% RSLogix 500 project Grain Separator - Onsite 24-11-05.RSS, saved by version 6.30.00.12 %
PROJECT "CORSON1"    % processor: SLC 500, 1747-L532 %

PROGRAM FILES
  LAD 2   10 rungs
  LAD 4   19 rungs
  LAD 5   124 rungs
  LAD 6   61 rungs
  LAD 7   60 rungs
  LAD 8   20 rungs
  LAD 9   20 rungs
  LAD 10   62 rungs
  LAD 11   79 rungs

DATA FILES
  O0 OUTPUT  11 elements
  I1 INPUT  11 elements
  S2 STATUS  83 elements
  B3 BINARY  1 elements
  T4 TIMER  1 elements
  C5 COUNTER  1 elements
  R6 CONTROL  1 elements
  N7 INTEGER  1 elements
  F8 FLOAT  1 elements
  B9   1 elements
  B10   2 elements
  T11   10 elements
  N12   1 elements
  B13   14 elements
  T14   60 elements
  N15   10 elements
  B16   5 elements
  T17   60 elements
  N18   1 elements
  B19   5 elements
  T20   60 elements
  N21   1 elements
  B22   5 elements
  T23   17 elements
  N24   1 elements
  B25   5 elements
  T26   16 elements
  N27   1 elements
  B28   1 elements
  T29   13 elements
  N30   1 elements
  B31   1 elements

LADDER 2
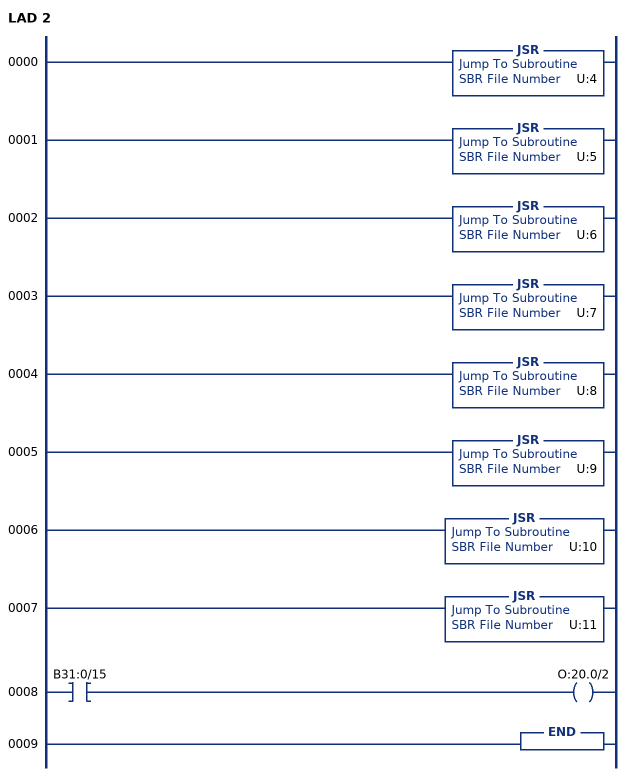
% Rung: 0 %
SOR JSR U:4 EOR
% Rung: 1 %
SOR JSR U:5 EOR
% Rung: 2 %
SOR JSR U:6 EOR
% Rung: 3 %
SOR JSR U:7 EOR
% Rung: 4 %
SOR JSR U:8 EOR
% Rung: 5 %
SOR JSR U:9 EOR
% Rung: 6 %
SOR JSR U:10 EOR
% Rung: 7 %
SOR JSR U:11 EOR
% Rung: 8 %
SOR XIC B31:0/15 OTE O:20.0/2 EOR
% Rung: 9 %
SOR END EOR

LADDER 4
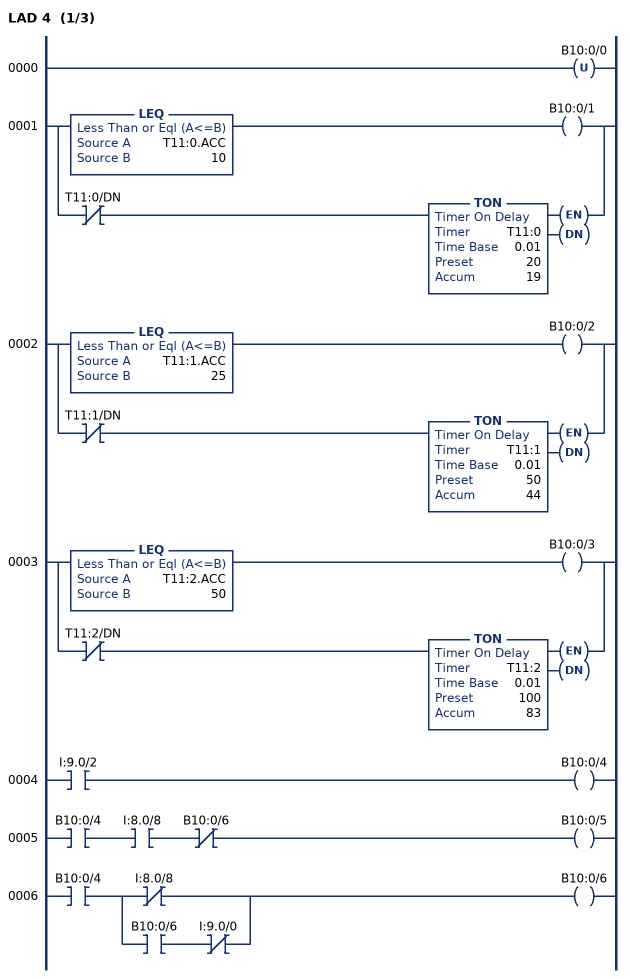
% Rung: 0 %
SOR OTU B10:0/0 EOR
% Rung: 1 %
SOR BST LEQ T11:0.ACC 10 OTE B10:0/1 NXB XIO T11:0/DN TON T11:0 0.01 20 19 BND EOR
% Rung: 2 %
SOR BST LEQ T11:1.ACC 25 OTE B10:0/2 NXB XIO T11:1/DN TON T11:1 0.01 50 44 BND EOR
% Rung: 3 %
SOR BST LEQ T11:2.ACC 50 OTE B10:0/3 NXB XIO T11:2/DN TON T11:2 0.01 100 83 BND EOR
% Rung: 4 %
SOR XIC I:9.0/2 OTE B10:0/4 EOR
% Rung: 5 %
SOR XIC B10:0/4 XIC I:8.0/8 XIO B10:0/6 OTE B10:0/5 EOR
% Rung: 6 %
SOR XIC B10:0/4 BST XIO I:8.0/8 NXB XIC B10:0/6 XIO I:9.0/0 BND OTE B10:0/6 EOR

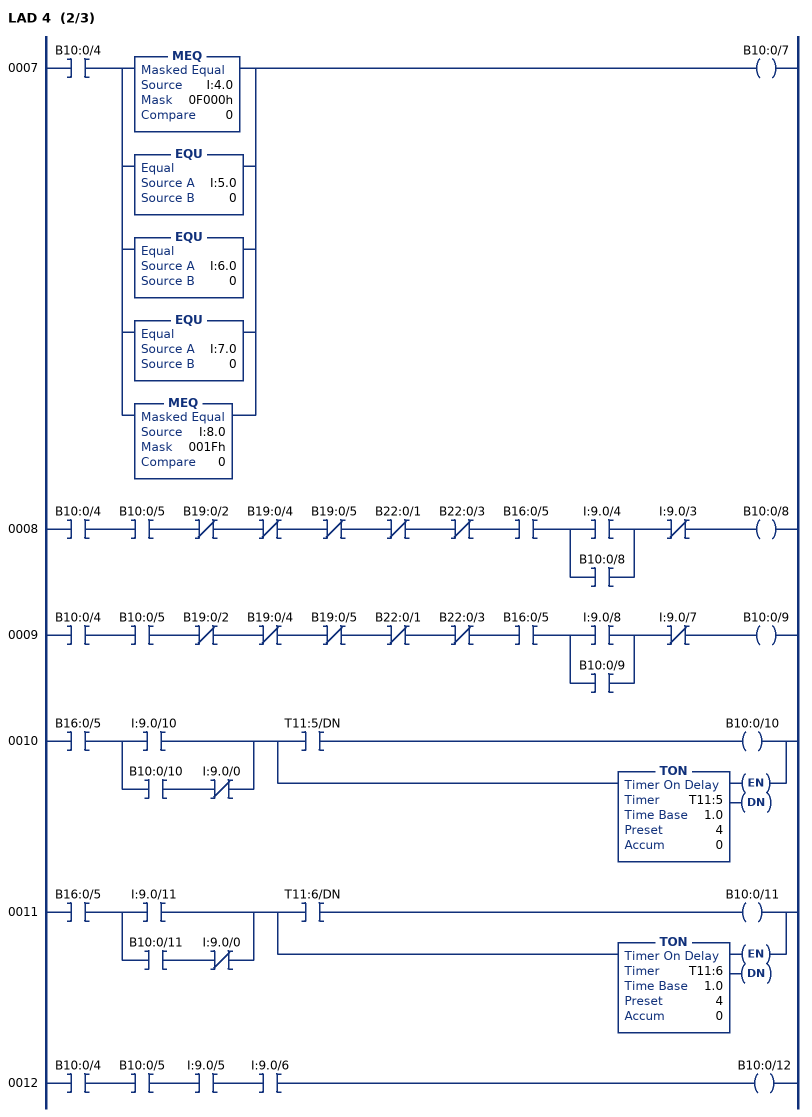
% Rung: 7 %
SOR XIC B10:0/4 BST MEQ I:4.0 0F000h 0 NXB EQU I:5.0 0 NXB EQU I:6.0 0 NXB EQU I:7.0 0 NXB MEQ I:8.0 001Fh 0 BND OTE B10:0/7 EOR
% Rung: 8 %
SOR XIC B10:0/4 XIC B10:0/5 XIO B19:0/2 XIO B19:0/4 XIO B19:0/5 XIO B22:0/1 XIO B22:0/3 XIC B16:0/5 BST XIC I:9.0/4 NXB XIC B10:0/8 BND XIO I:9.0/3 OTE B10:0/8 EOR
% Rung: 9 %
SOR XIC B10:0/4 XIC B10:0/5 XIO B19:0/2 XIO B19:0/4 XIO B19:0/5 XIO B22:0/1 XIO B22:0/3 XIC B16:0/5 BST XIC I:9.0/8 NXB XIC B10:0/9 BND XIO I:9.0/7 OTE B10:0/9 EOR
% Rung: 10 %
SOR XIC B16:0/5 BST XIC I:9.0/10 NXB XIC B10:0/10 XIO I:9.0/0 BND BST XIC T11:5/DN OTE B10:0/10 NXB TON T11:5 1.0 4 0 BND EOR
% Rung: 11 %
SOR XIC B16:0/5 BST XIC I:9.0/11 NXB XIC B10:0/11 XIO I:9.0/0 BND BST XIC T11:6/DN OTE B10:0/11 NXB TON T11:6 1.0 4 0 BND EOR
% Rung: 12 %
SOR XIC B10:0/4 XIC B10:0/5 XIC I:9.0/5 XIC I:9.0/6 OTE B10:0/12 EOR

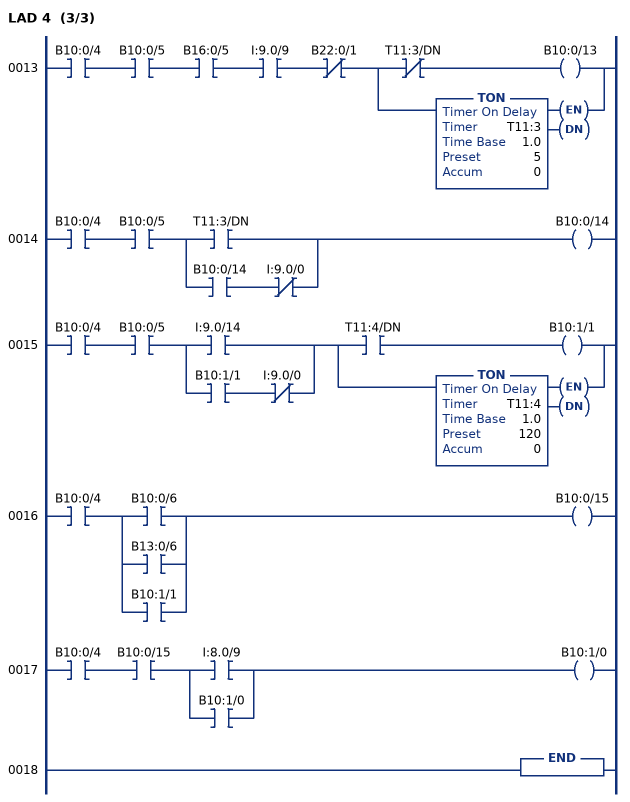
% Rung: 13 %
SOR XIC B10:0/4 XIC B10:0/5 XIC B16:0/5 XIC I:9.0/9 XIO B22:0/1 BST XIO T11:3/DN OTE B10:0/13 NXB TON T11:3 1.0 5 0 BND EOR
% Rung: 14 %
SOR XIC B10:0/4 XIC B10:0/5 BST XIC T11:3/DN NXB XIC B10:0/14 XIO I:9.0/0 BND OTE B10:0/14 EOR
% Rung: 15 %
SOR XIC B10:0/4 XIC B10:0/5 BST XIC I:9.0/14 NXB XIC B10:1/1 XIO I:9.0/0 BND BST XIC T11:4/DN OTE B10:1/1 NXB TON T11:4 1.0 120 0 BND EOR
% Rung: 16 %
SOR XIC B10:0/4 BST XIC B10:0/6 NXB XIC B13:0/6 NXB XIC B10:1/1 BND OTE B10:0/15 EOR
% Rung: 17 %
SOR XIC B10:0/4 XIC B10:0/15 BST XIC I:8.0/9 NXB XIC B10:1/0 BND OTE B10:1/0 EOR
% Rung: 18 %
SOR END EOR

LADDER 5
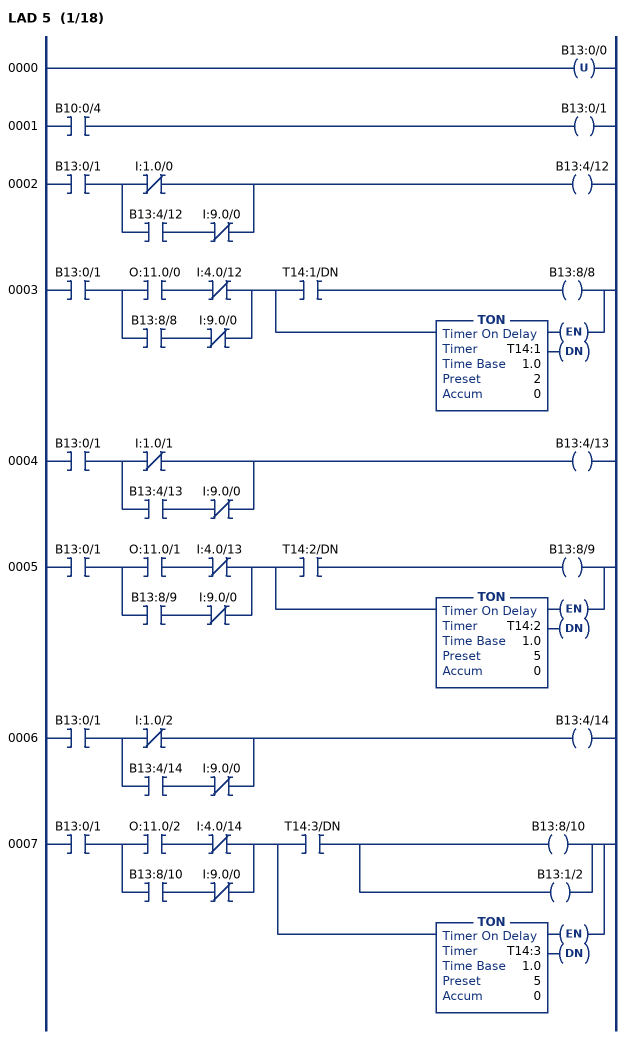
% Rung: 0 %
SOR OTU B13:0/0 EOR
% Rung: 1 %
SOR XIC B10:0/4 OTE B13:0/1 EOR
% Rung: 2 %
SOR XIC B13:0/1 BST XIO I:1.0/0 NXB XIC B13:4/12 XIO I:9.0/0 BND OTE B13:4/12 EOR
% Rung: 3 %
SOR XIC B13:0/1 BST XIC O:11.0/0 XIO I:4.0/12 NXB XIC B13:8/8 XIO I:9.0/0 BND BST XIC T14:1/DN OTE B13:8/8 NXB TON T14:1 1.0 2 0 BND EOR
% Rung: 4 %
SOR XIC B13:0/1 BST XIO I:1.0/1 NXB XIC B13:4/13 XIO I:9.0/0 BND OTE B13:4/13 EOR
% Rung: 5 %
SOR XIC B13:0/1 BST XIC O:11.0/1 XIO I:4.0/13 NXB XIC B13:8/9 XIO I:9.0/0 BND BST XIC T14:2/DN OTE B13:8/9 NXB TON T14:2 1.0 5 0 BND EOR
% Rung: 6 %
SOR XIC B13:0/1 BST XIO I:1.0/2 NXB XIC B13:4/14 XIO I:9.0/0 BND OTE B13:4/14 EOR
% Rung: 7 %
SOR XIC B13:0/1 BST XIC O:11.0/2 XIO I:4.0/14 NXB XIC B13:8/10 XIO I:9.0/0 BND BST XIC T14:3/DN BST OTE B13:8/10 NXB OTE B13:1/2 BND NXB TON T14:3 1.0 5 0 BND EOR

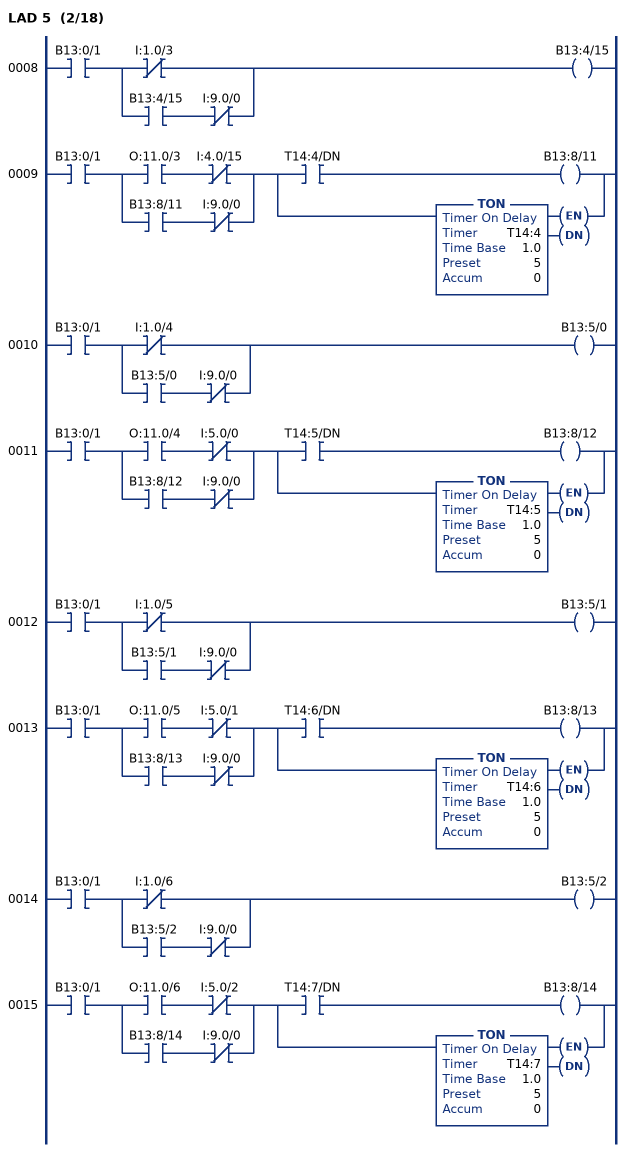
% Rung: 8 %
SOR XIC B13:0/1 BST XIO I:1.0/3 NXB XIC B13:4/15 XIO I:9.0/0 BND OTE B13:4/15 EOR
% Rung: 9 %
SOR XIC B13:0/1 BST XIC O:11.0/3 XIO I:4.0/15 NXB XIC B13:8/11 XIO I:9.0/0 BND BST XIC T14:4/DN OTE B13:8/11 NXB TON T14:4 1.0 5 0 BND EOR
% Rung: 10 %
SOR XIC B13:0/1 BST XIO I:1.0/4 NXB XIC B13:5/0 XIO I:9.0/0 BND OTE B13:5/0 EOR
% Rung: 11 %
SOR XIC B13:0/1 BST XIC O:11.0/4 XIO I:5.0/0 NXB XIC B13:8/12 XIO I:9.0/0 BND BST XIC T14:5/DN OTE B13:8/12 NXB TON T14:5 1.0 5 0 BND EOR
% Rung: 12 %
SOR XIC B13:0/1 BST XIO I:1.0/5 NXB XIC B13:5/1 XIO I:9.0/0 BND OTE B13:5/1 EOR
% Rung: 13 %
SOR XIC B13:0/1 BST XIC O:11.0/5 XIO I:5.0/1 NXB XIC B13:8/13 XIO I:9.0/0 BND BST XIC T14:6/DN OTE B13:8/13 NXB TON T14:6 1.0 5 0 BND EOR
% Rung: 14 %
SOR XIC B13:0/1 BST XIO I:1.0/6 NXB XIC B13:5/2 XIO I:9.0/0 BND OTE B13:5/2 EOR
% Rung: 15 %
SOR XIC B13:0/1 BST XIC O:11.0/6 XIO I:5.0/2 NXB XIC B13:8/14 XIO I:9.0/0 BND BST XIC T14:7/DN OTE B13:8/14 NXB TON T14:7 1.0 5 0 BND EOR

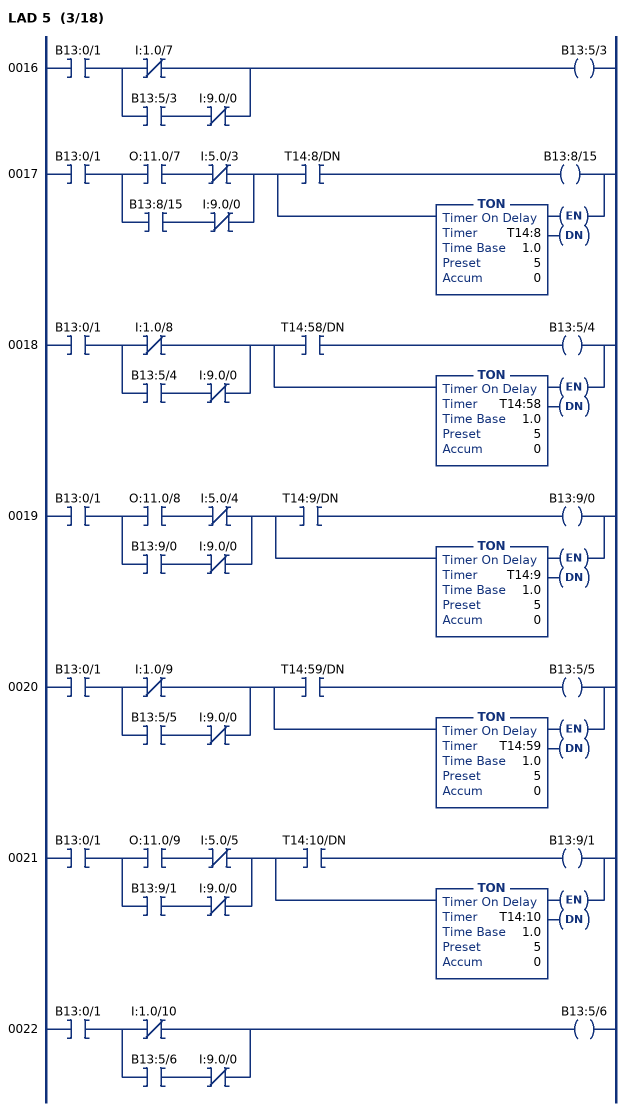
% Rung: 16 %
SOR XIC B13:0/1 BST XIO I:1.0/7 NXB XIC B13:5/3 XIO I:9.0/0 BND OTE B13:5/3 EOR
% Rung: 17 %
SOR XIC B13:0/1 BST XIC O:11.0/7 XIO I:5.0/3 NXB XIC B13:8/15 XIO I:9.0/0 BND BST XIC T14:8/DN OTE B13:8/15 NXB TON T14:8 1.0 5 0 BND EOR
% Rung: 18 %
SOR XIC B13:0/1 BST XIO I:1.0/8 NXB XIC B13:5/4 XIO I:9.0/0 BND BST XIC T14:58/DN OTE B13:5/4 NXB TON T14:58 1.0 5 0 BND EOR
% Rung: 19 %
SOR XIC B13:0/1 BST XIC O:11.0/8 XIO I:5.0/4 NXB XIC B13:9/0 XIO I:9.0/0 BND BST XIC T14:9/DN OTE B13:9/0 NXB TON T14:9 1.0 5 0 BND EOR
% Rung: 20 %
SOR XIC B13:0/1 BST XIO I:1.0/9 NXB XIC B13:5/5 XIO I:9.0/0 BND BST XIC T14:59/DN OTE B13:5/5 NXB TON T14:59 1.0 5 0 BND EOR
% Rung: 21 %
SOR XIC B13:0/1 BST XIC O:11.0/9 XIO I:5.0/5 NXB XIC B13:9/1 XIO I:9.0/0 BND BST XIC T14:10/DN OTE B13:9/1 NXB TON T14:10 1.0 5 0 BND EOR
% Rung: 22 %
SOR XIC B13:0/1 BST XIO I:1.0/10 NXB XIC B13:5/6 XIO I:9.0/0 BND OTE B13:5/6 EOR

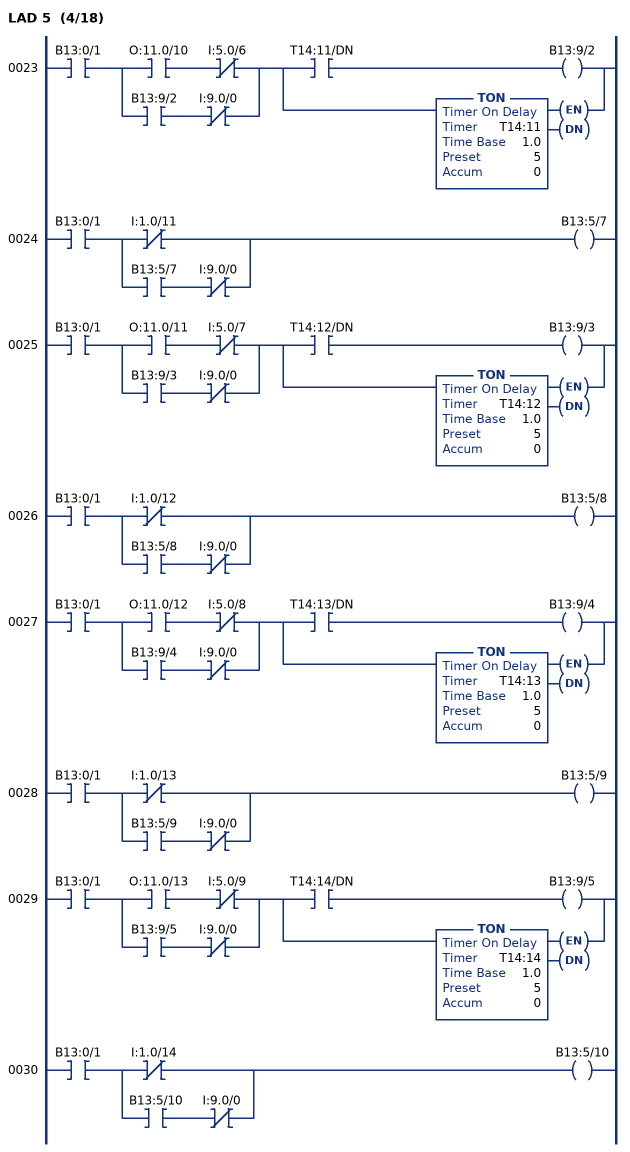
% Rung: 23 %
SOR XIC B13:0/1 BST XIC O:11.0/10 XIO I:5.0/6 NXB XIC B13:9/2 XIO I:9.0/0 BND BST XIC T14:11/DN OTE B13:9/2 NXB TON T14:11 1.0 5 0 BND EOR
% Rung: 24 %
SOR XIC B13:0/1 BST XIO I:1.0/11 NXB XIC B13:5/7 XIO I:9.0/0 BND OTE B13:5/7 EOR
% Rung: 25 %
SOR XIC B13:0/1 BST XIC O:11.0/11 XIO I:5.0/7 NXB XIC B13:9/3 XIO I:9.0/0 BND BST XIC T14:12/DN OTE B13:9/3 NXB TON T14:12 1.0 5 0 BND EOR
% Rung: 26 %
SOR XIC B13:0/1 BST XIO I:1.0/12 NXB XIC B13:5/8 XIO I:9.0/0 BND OTE B13:5/8 EOR
% Rung: 27 %
SOR XIC B13:0/1 BST XIC O:11.0/12 XIO I:5.0/8 NXB XIC B13:9/4 XIO I:9.0/0 BND BST XIC T14:13/DN OTE B13:9/4 NXB TON T14:13 1.0 5 0 BND EOR
% Rung: 28 %
SOR XIC B13:0/1 BST XIO I:1.0/13 NXB XIC B13:5/9 XIO I:9.0/0 BND OTE B13:5/9 EOR
% Rung: 29 %
SOR XIC B13:0/1 BST XIC O:11.0/13 XIO I:5.0/9 NXB XIC B13:9/5 XIO I:9.0/0 BND BST XIC T14:14/DN OTE B13:9/5 NXB TON T14:14 1.0 5 0 BND EOR
% Rung: 30 %
SOR XIC B13:0/1 BST XIO I:1.0/14 NXB XIC B13:5/10 XIO I:9.0/0 BND OTE B13:5/10 EOR

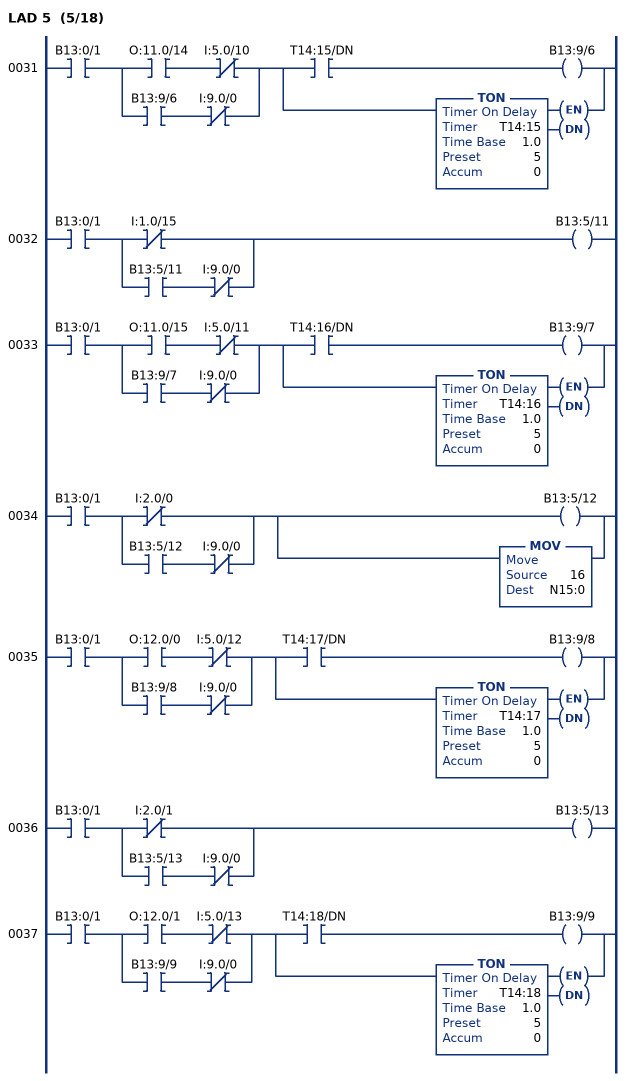
% Rung: 31 %
SOR XIC B13:0/1 BST XIC O:11.0/14 XIO I:5.0/10 NXB XIC B13:9/6 XIO I:9.0/0 BND BST XIC T14:15/DN OTE B13:9/6 NXB TON T14:15 1.0 5 0 BND EOR
% Rung: 32 %
SOR XIC B13:0/1 BST XIO I:1.0/15 NXB XIC B13:5/11 XIO I:9.0/0 BND OTE B13:5/11 EOR
% Rung: 33 %
SOR XIC B13:0/1 BST XIC O:11.0/15 XIO I:5.0/11 NXB XIC B13:9/7 XIO I:9.0/0 BND BST XIC T14:16/DN OTE B13:9/7 NXB TON T14:16 1.0 5 0 BND EOR
% Rung: 34 %
SOR XIC B13:0/1 BST XIO I:2.0/0 NXB XIC B13:5/12 XIO I:9.0/0 BND BST OTE B13:5/12 NXB MOV 16 N15:0 BND EOR
% Rung: 35 %
SOR XIC B13:0/1 BST XIC O:12.0/0 XIO I:5.0/12 NXB XIC B13:9/8 XIO I:9.0/0 BND BST XIC T14:17/DN OTE B13:9/8 NXB TON T14:17 1.0 5 0 BND EOR
% Rung: 36 %
SOR XIC B13:0/1 BST XIO I:2.0/1 NXB XIC B13:5/13 XIO I:9.0/0 BND OTE B13:5/13 EOR
% Rung: 37 %
SOR XIC B13:0/1 BST XIC O:12.0/1 XIO I:5.0/13 NXB XIC B13:9/9 XIO I:9.0/0 BND BST XIC T14:18/DN OTE B13:9/9 NXB TON T14:18 1.0 5 0 BND EOR

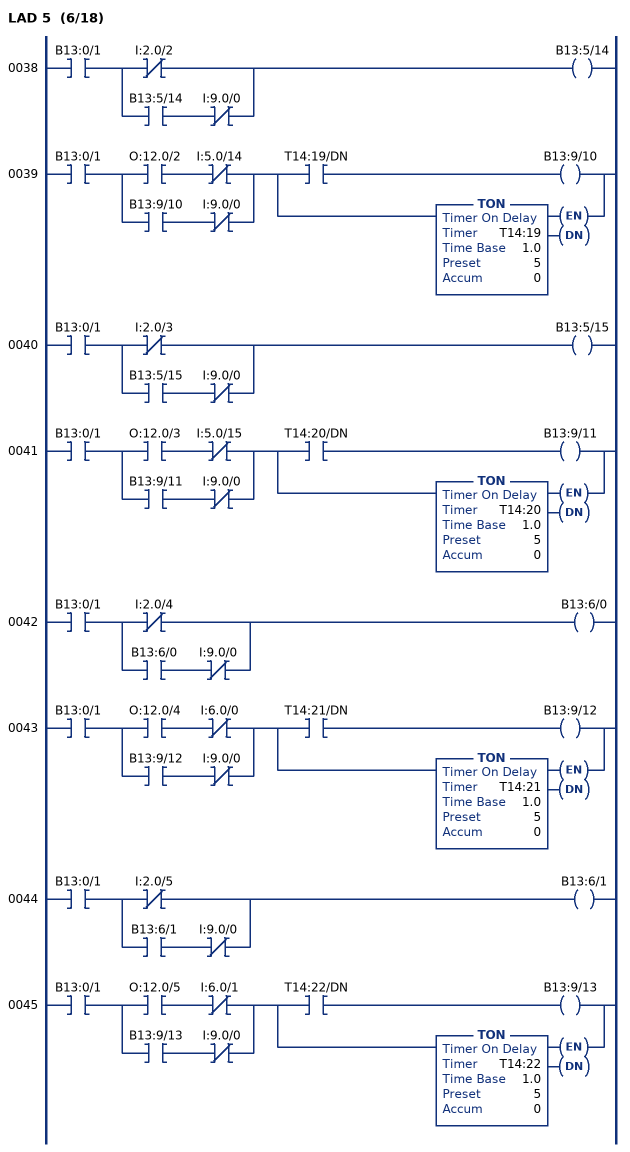
% Rung: 38 %
SOR XIC B13:0/1 BST XIO I:2.0/2 NXB XIC B13:5/14 XIO I:9.0/0 BND OTE B13:5/14 EOR
% Rung: 39 %
SOR XIC B13:0/1 BST XIC O:12.0/2 XIO I:5.0/14 NXB XIC B13:9/10 XIO I:9.0/0 BND BST XIC T14:19/DN OTE B13:9/10 NXB TON T14:19 1.0 5 0 BND EOR
% Rung: 40 %
SOR XIC B13:0/1 BST XIO I:2.0/3 NXB XIC B13:5/15 XIO I:9.0/0 BND OTE B13:5/15 EOR
% Rung: 41 %
SOR XIC B13:0/1 BST XIC O:12.0/3 XIO I:5.0/15 NXB XIC B13:9/11 XIO I:9.0/0 BND BST XIC T14:20/DN OTE B13:9/11 NXB TON T14:20 1.0 5 0 BND EOR
% Rung: 42 %
SOR XIC B13:0/1 BST XIO I:2.0/4 NXB XIC B13:6/0 XIO I:9.0/0 BND OTE B13:6/0 EOR
% Rung: 43 %
SOR XIC B13:0/1 BST XIC O:12.0/4 XIO I:6.0/0 NXB XIC B13:9/12 XIO I:9.0/0 BND BST XIC T14:21/DN OTE B13:9/12 NXB TON T14:21 1.0 5 0 BND EOR
% Rung: 44 %
SOR XIC B13:0/1 BST XIO I:2.0/5 NXB XIC B13:6/1 XIO I:9.0/0 BND OTE B13:6/1 EOR
% Rung: 45 %
SOR XIC B13:0/1 BST XIC O:12.0/5 XIO I:6.0/1 NXB XIC B13:9/13 XIO I:9.0/0 BND BST XIC T14:22/DN OTE B13:9/13 NXB TON T14:22 1.0 5 0 BND EOR

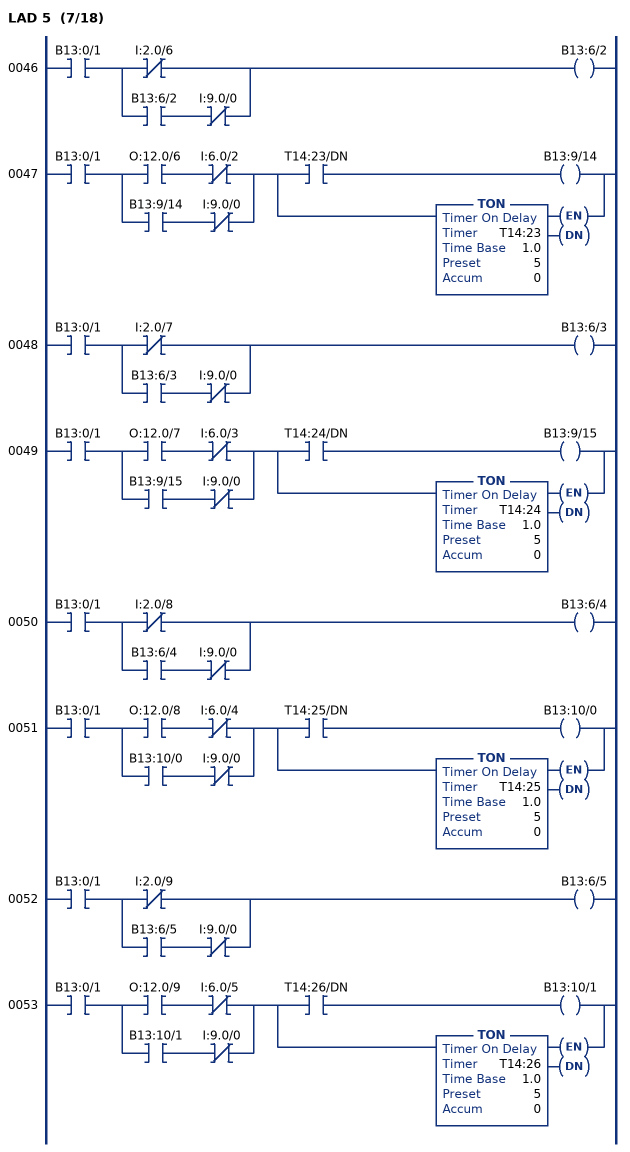
% Rung: 46 %
SOR XIC B13:0/1 BST XIO I:2.0/6 NXB XIC B13:6/2 XIO I:9.0/0 BND OTE B13:6/2 EOR
% Rung: 47 %
SOR XIC B13:0/1 BST XIC O:12.0/6 XIO I:6.0/2 NXB XIC B13:9/14 XIO I:9.0/0 BND BST XIC T14:23/DN OTE B13:9/14 NXB TON T14:23 1.0 5 0 BND EOR
% Rung: 48 %
SOR XIC B13:0/1 BST XIO I:2.0/7 NXB XIC B13:6/3 XIO I:9.0/0 BND OTE B13:6/3 EOR
% Rung: 49 %
SOR XIC B13:0/1 BST XIC O:12.0/7 XIO I:6.0/3 NXB XIC B13:9/15 XIO I:9.0/0 BND BST XIC T14:24/DN OTE B13:9/15 NXB TON T14:24 1.0 5 0 BND EOR
% Rung: 50 %
SOR XIC B13:0/1 BST XIO I:2.0/8 NXB XIC B13:6/4 XIO I:9.0/0 BND OTE B13:6/4 EOR
% Rung: 51 %
SOR XIC B13:0/1 BST XIC O:12.0/8 XIO I:6.0/4 NXB XIC B13:10/0 XIO I:9.0/0 BND BST XIC T14:25/DN OTE B13:10/0 NXB TON T14:25 1.0 5 0 BND EOR
% Rung: 52 %
SOR XIC B13:0/1 BST XIO I:2.0/9 NXB XIC B13:6/5 XIO I:9.0/0 BND OTE B13:6/5 EOR
% Rung: 53 %
SOR XIC B13:0/1 BST XIC O:12.0/9 XIO I:6.0/5 NXB XIC B13:10/1 XIO I:9.0/0 BND BST XIC T14:26/DN OTE B13:10/1 NXB TON T14:26 1.0 5 0 BND EOR

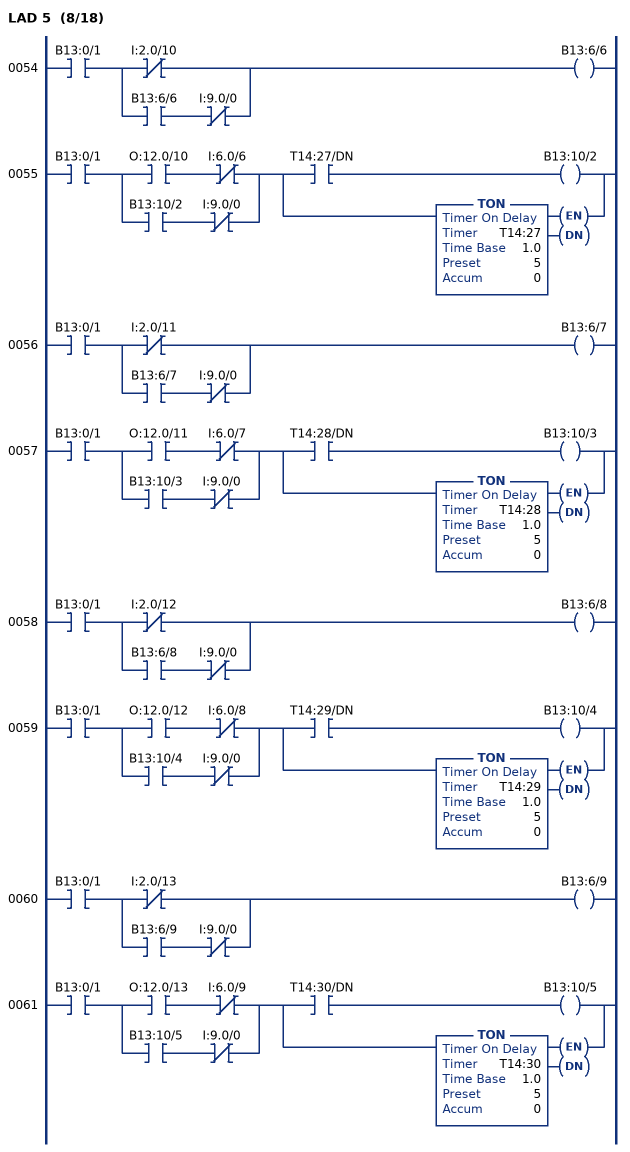
% Rung: 54 %
SOR XIC B13:0/1 BST XIO I:2.0/10 NXB XIC B13:6/6 XIO I:9.0/0 BND OTE B13:6/6 EOR
% Rung: 55 %
SOR XIC B13:0/1 BST XIC O:12.0/10 XIO I:6.0/6 NXB XIC B13:10/2 XIO I:9.0/0 BND BST XIC T14:27/DN OTE B13:10/2 NXB TON T14:27 1.0 5 0 BND EOR
% Rung: 56 %
SOR XIC B13:0/1 BST XIO I:2.0/11 NXB XIC B13:6/7 XIO I:9.0/0 BND OTE B13:6/7 EOR
% Rung: 57 %
SOR XIC B13:0/1 BST XIC O:12.0/11 XIO I:6.0/7 NXB XIC B13:10/3 XIO I:9.0/0 BND BST XIC T14:28/DN OTE B13:10/3 NXB TON T14:28 1.0 5 0 BND EOR
% Rung: 58 %
SOR XIC B13:0/1 BST XIO I:2.0/12 NXB XIC B13:6/8 XIO I:9.0/0 BND OTE B13:6/8 EOR
% Rung: 59 %
SOR XIC B13:0/1 BST XIC O:12.0/12 XIO I:6.0/8 NXB XIC B13:10/4 XIO I:9.0/0 BND BST XIC T14:29/DN OTE B13:10/4 NXB TON T14:29 1.0 5 0 BND EOR
% Rung: 60 %
SOR XIC B13:0/1 BST XIO I:2.0/13 NXB XIC B13:6/9 XIO I:9.0/0 BND OTE B13:6/9 EOR
% Rung: 61 %
SOR XIC B13:0/1 BST XIC O:12.0/13 XIO I:6.0/9 NXB XIC B13:10/5 XIO I:9.0/0 BND BST XIC T14:30/DN OTE B13:10/5 NXB TON T14:30 1.0 5 0 BND EOR

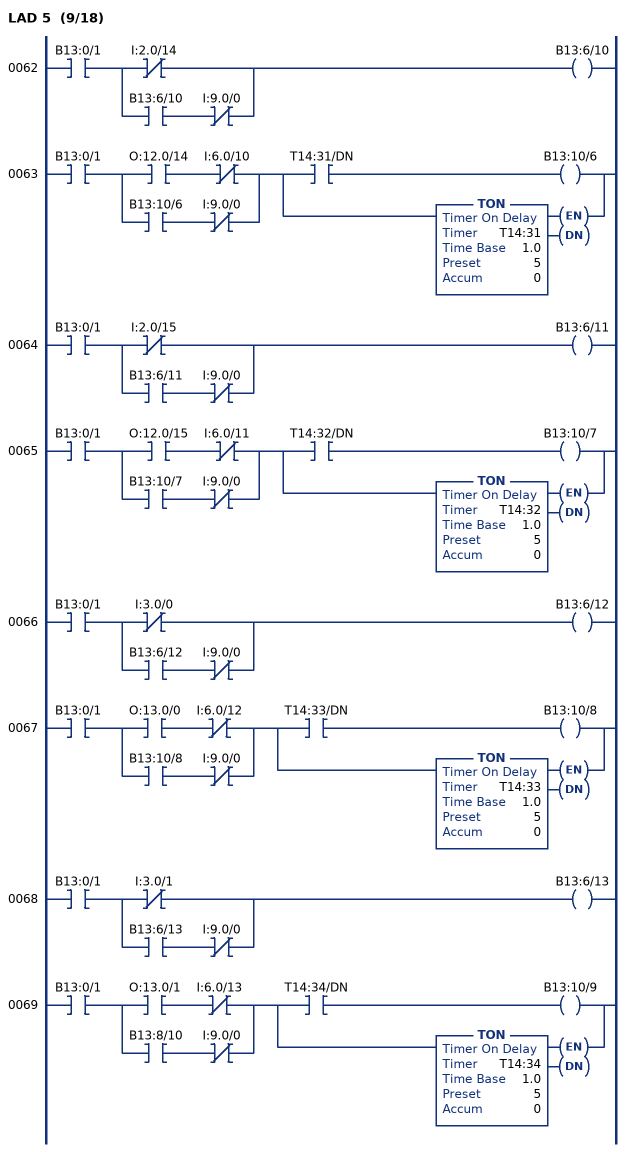
% Rung: 62 %
SOR XIC B13:0/1 BST XIO I:2.0/14 NXB XIC B13:6/10 XIO I:9.0/0 BND OTE B13:6/10 EOR
% Rung: 63 %
SOR XIC B13:0/1 BST XIC O:12.0/14 XIO I:6.0/10 NXB XIC B13:10/6 XIO I:9.0/0 BND BST XIC T14:31/DN OTE B13:10/6 NXB TON T14:31 1.0 5 0 BND EOR
% Rung: 64 %
SOR XIC B13:0/1 BST XIO I:2.0/15 NXB XIC B13:6/11 XIO I:9.0/0 BND OTE B13:6/11 EOR
% Rung: 65 %
SOR XIC B13:0/1 BST XIC O:12.0/15 XIO I:6.0/11 NXB XIC B13:10/7 XIO I:9.0/0 BND BST XIC T14:32/DN OTE B13:10/7 NXB TON T14:32 1.0 5 0 BND EOR
% Rung: 66 %
SOR XIC B13:0/1 BST XIO I:3.0/0 NXB XIC B13:6/12 XIO I:9.0/0 BND OTE B13:6/12 EOR
% Rung: 67 %
SOR XIC B13:0/1 BST XIC O:13.0/0 XIO I:6.0/12 NXB XIC B13:10/8 XIO I:9.0/0 BND BST XIC T14:33/DN OTE B13:10/8 NXB TON T14:33 1.0 5 0 BND EOR
% Rung: 68 %
SOR XIC B13:0/1 BST XIO I:3.0/1 NXB XIC B13:6/13 XIO I:9.0/0 BND OTE B13:6/13 EOR
% Rung: 69 %
SOR XIC B13:0/1 BST XIC O:13.0/1 XIO I:6.0/13 NXB XIC B13:8/10 XIO I:9.0/0 BND BST XIC T14:34/DN OTE B13:10/9 NXB TON T14:34 1.0 5 0 BND EOR

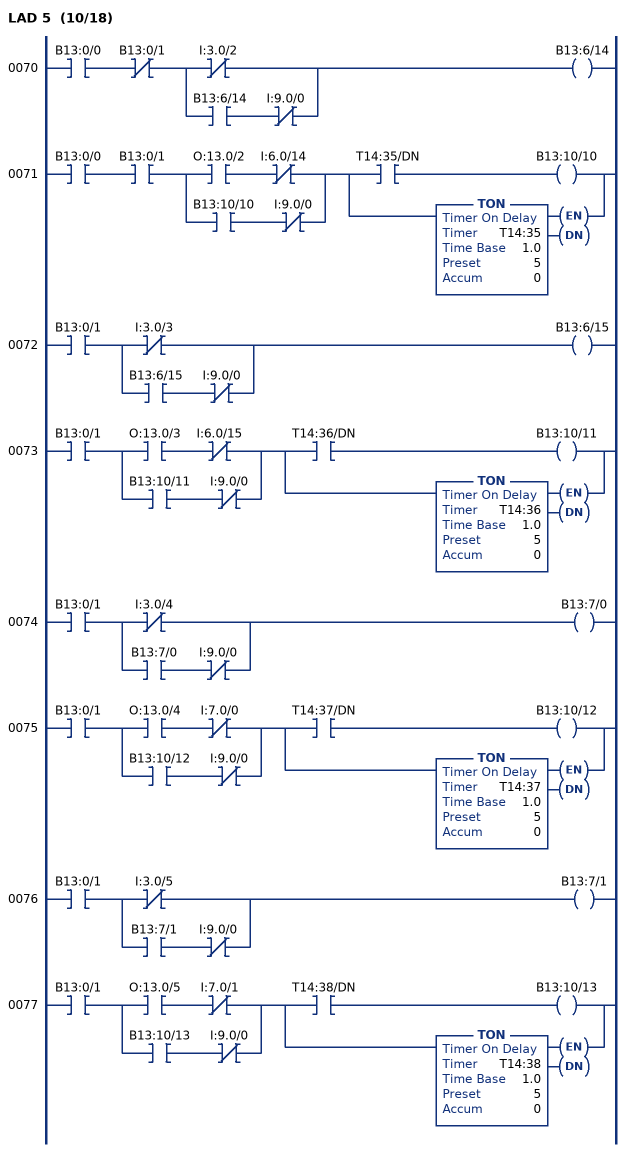
% Rung: 70 %
SOR XIC B13:0/0 XIO B13:0/1 BST XIO I:3.0/2 NXB XIC B13:6/14 XIO I:9.0/0 BND OTE B13:6/14 EOR
% Rung: 71 %
SOR XIC B13:0/0 XIC B13:0/1 BST XIC O:13.0/2 XIO I:6.0/14 NXB XIC B13:10/10 XIO I:9.0/0 BND BST XIC T14:35/DN OTE B13:10/10 NXB TON T14:35 1.0 5 0 BND EOR
% Rung: 72 %
SOR XIC B13:0/1 BST XIO I:3.0/3 NXB XIC B13:6/15 XIO I:9.0/0 BND OTE B13:6/15 EOR
% Rung: 73 %
SOR XIC B13:0/1 BST XIC O:13.0/3 XIO I:6.0/15 NXB XIC B13:10/11 XIO I:9.0/0 BND BST XIC T14:36/DN OTE B13:10/11 NXB TON T14:36 1.0 5 0 BND EOR
% Rung: 74 %
SOR XIC B13:0/1 BST XIO I:3.0/4 NXB XIC B13:7/0 XIO I:9.0/0 BND OTE B13:7/0 EOR
% Rung: 75 %
SOR XIC B13:0/1 BST XIC O:13.0/4 XIO I:7.0/0 NXB XIC B13:10/12 XIO I:9.0/0 BND BST XIC T14:37/DN OTE B13:10/12 NXB TON T14:37 1.0 5 0 BND EOR
% Rung: 76 %
SOR XIC B13:0/1 BST XIO I:3.0/5 NXB XIC B13:7/1 XIO I:9.0/0 BND OTE B13:7/1 EOR
% Rung: 77 %
SOR XIC B13:0/1 BST XIC O:13.0/5 XIO I:7.0/1 NXB XIC B13:10/13 XIO I:9.0/0 BND BST XIC T14:38/DN OTE B13:10/13 NXB TON T14:38 1.0 5 0 BND EOR

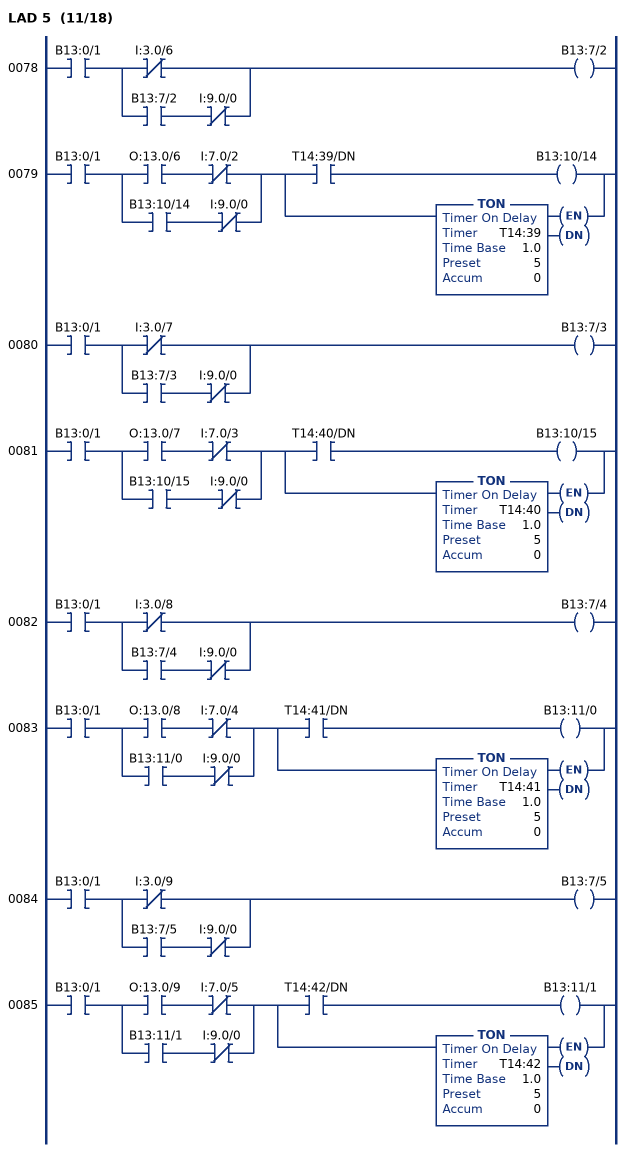
% Rung: 78 %
SOR XIC B13:0/1 BST XIO I:3.0/6 NXB XIC B13:7/2 XIO I:9.0/0 BND OTE B13:7/2 EOR
% Rung: 79 %
SOR XIC B13:0/1 BST XIC O:13.0/6 XIO I:7.0/2 NXB XIC B13:10/14 XIO I:9.0/0 BND BST XIC T14:39/DN OTE B13:10/14 NXB TON T14:39 1.0 5 0 BND EOR
% Rung: 80 %
SOR XIC B13:0/1 BST XIO I:3.0/7 NXB XIC B13:7/3 XIO I:9.0/0 BND OTE B13:7/3 EOR
% Rung: 81 %
SOR XIC B13:0/1 BST XIC O:13.0/7 XIO I:7.0/3 NXB XIC B13:10/15 XIO I:9.0/0 BND BST XIC T14:40/DN OTE B13:10/15 NXB TON T14:40 1.0 5 0 BND EOR
% Rung: 82 %
SOR XIC B13:0/1 BST XIO I:3.0/8 NXB XIC B13:7/4 XIO I:9.0/0 BND OTE B13:7/4 EOR
% Rung: 83 %
SOR XIC B13:0/1 BST XIC O:13.0/8 XIO I:7.0/4 NXB XIC B13:11/0 XIO I:9.0/0 BND BST XIC T14:41/DN OTE B13:11/0 NXB TON T14:41 1.0 5 0 BND EOR
% Rung: 84 %
SOR XIC B13:0/1 BST XIO I:3.0/9 NXB XIC B13:7/5 XIO I:9.0/0 BND OTE B13:7/5 EOR
% Rung: 85 %
SOR XIC B13:0/1 BST XIC O:13.0/9 XIO I:7.0/5 NXB XIC B13:11/1 XIO I:9.0/0 BND BST XIC T14:42/DN OTE B13:11/1 NXB TON T14:42 1.0 5 0 BND EOR

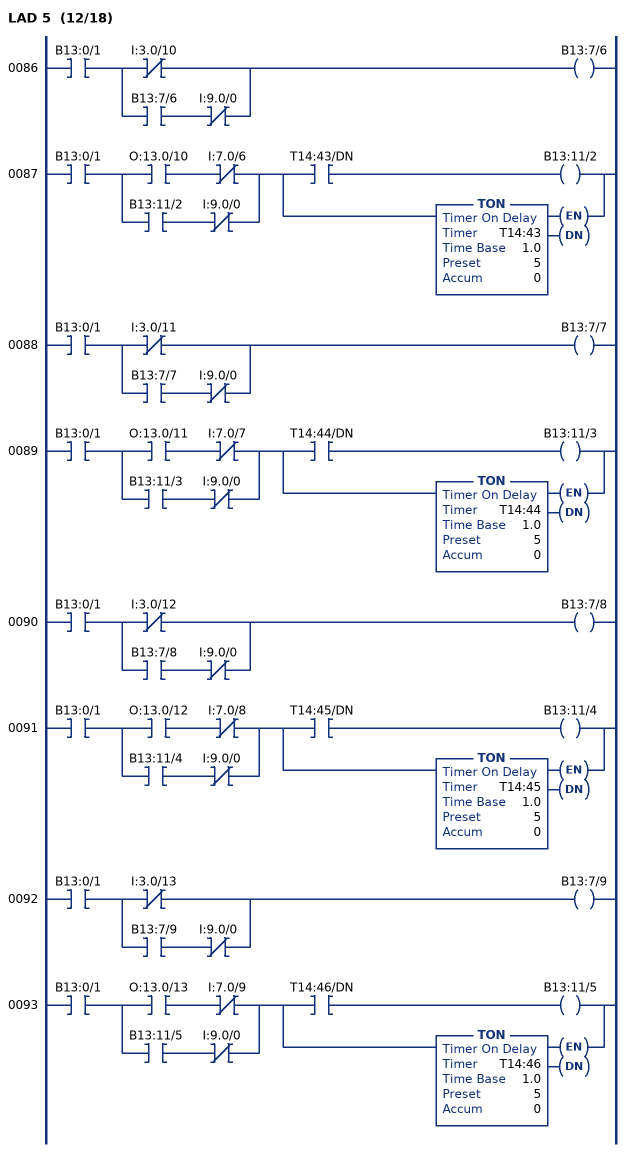
% Rung: 86 %
SOR XIC B13:0/1 BST XIO I:3.0/10 NXB XIC B13:7/6 XIO I:9.0/0 BND OTE B13:7/6 EOR
% Rung: 87 %
SOR XIC B13:0/1 BST XIC O:13.0/10 XIO I:7.0/6 NXB XIC B13:11/2 XIO I:9.0/0 BND BST XIC T14:43/DN OTE B13:11/2 NXB TON T14:43 1.0 5 0 BND EOR
% Rung: 88 %
SOR XIC B13:0/1 BST XIO I:3.0/11 NXB XIC B13:7/7 XIO I:9.0/0 BND OTE B13:7/7 EOR
% Rung: 89 %
SOR XIC B13:0/1 BST XIC O:13.0/11 XIO I:7.0/7 NXB XIC B13:11/3 XIO I:9.0/0 BND BST XIC T14:44/DN OTE B13:11/3 NXB TON T14:44 1.0 5 0 BND EOR
% Rung: 90 %
SOR XIC B13:0/1 BST XIO I:3.0/12 NXB XIC B13:7/8 XIO I:9.0/0 BND OTE B13:7/8 EOR
% Rung: 91 %
SOR XIC B13:0/1 BST XIC O:13.0/12 XIO I:7.0/8 NXB XIC B13:11/4 XIO I:9.0/0 BND BST XIC T14:45/DN OTE B13:11/4 NXB TON T14:45 1.0 5 0 BND EOR
% Rung: 92 %
SOR XIC B13:0/1 BST XIO I:3.0/13 NXB XIC B13:7/9 XIO I:9.0/0 BND OTE B13:7/9 EOR
% Rung: 93 %
SOR XIC B13:0/1 BST XIC O:13.0/13 XIO I:7.0/9 NXB XIC B13:11/5 XIO I:9.0/0 BND BST XIC T14:46/DN OTE B13:11/5 NXB TON T14:46 1.0 5 0 BND EOR

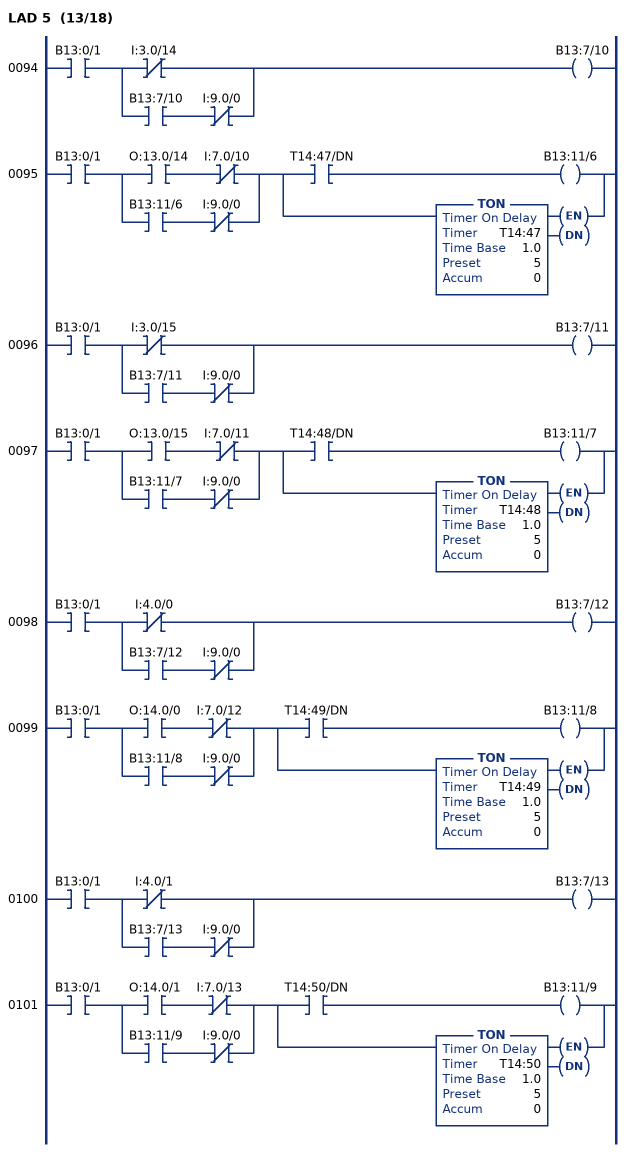
% Rung: 94 %
SOR XIC B13:0/1 BST XIO I:3.0/14 NXB XIC B13:7/10 XIO I:9.0/0 BND OTE B13:7/10 EOR
% Rung: 95 %
SOR XIC B13:0/1 BST XIC O:13.0/14 XIO I:7.0/10 NXB XIC B13:11/6 XIO I:9.0/0 BND BST XIC T14:47/DN OTE B13:11/6 NXB TON T14:47 1.0 5 0 BND EOR
% Rung: 96 %
SOR XIC B13:0/1 BST XIO I:3.0/15 NXB XIC B13:7/11 XIO I:9.0/0 BND OTE B13:7/11 EOR
% Rung: 97 %
SOR XIC B13:0/1 BST XIC O:13.0/15 XIO I:7.0/11 NXB XIC B13:11/7 XIO I:9.0/0 BND BST XIC T14:48/DN OTE B13:11/7 NXB TON T14:48 1.0 5 0 BND EOR
% Rung: 98 %
SOR XIC B13:0/1 BST XIO I:4.0/0 NXB XIC B13:7/12 XIO I:9.0/0 BND OTE B13:7/12 EOR
% Rung: 99 %
SOR XIC B13:0/1 BST XIC O:14.0/0 XIO I:7.0/12 NXB XIC B13:11/8 XIO I:9.0/0 BND BST XIC T14:49/DN OTE B13:11/8 NXB TON T14:49 1.0 5 0 BND EOR
% Rung: 100 %
SOR XIC B13:0/1 BST XIO I:4.0/1 NXB XIC B13:7/13 XIO I:9.0/0 BND OTE B13:7/13 EOR
% Rung: 101 %
SOR XIC B13:0/1 BST XIC O:14.0/1 XIO I:7.0/13 NXB XIC B13:11/9 XIO I:9.0/0 BND BST XIC T14:50/DN OTE B13:11/9 NXB TON T14:50 1.0 5 0 BND EOR

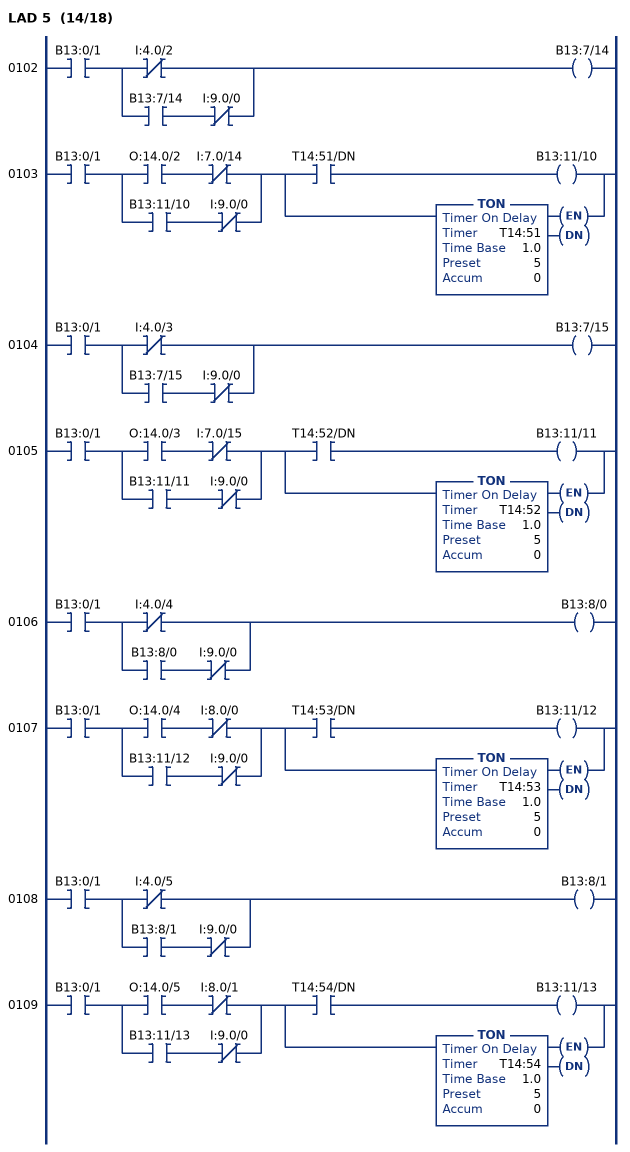
% Rung: 102 %
SOR XIC B13:0/1 BST XIO I:4.0/2 NXB XIC B13:7/14 XIO I:9.0/0 BND OTE B13:7/14 EOR
% Rung: 103 %
SOR XIC B13:0/1 BST XIC O:14.0/2 XIO I:7.0/14 NXB XIC B13:11/10 XIO I:9.0/0 BND BST XIC T14:51/DN OTE B13:11/10 NXB TON T14:51 1.0 5 0 BND EOR
% Rung: 104 %
SOR XIC B13:0/1 BST XIO I:4.0/3 NXB XIC B13:7/15 XIO I:9.0/0 BND OTE B13:7/15 EOR
% Rung: 105 %
SOR XIC B13:0/1 BST XIC O:14.0/3 XIO I:7.0/15 NXB XIC B13:11/11 XIO I:9.0/0 BND BST XIC T14:52/DN OTE B13:11/11 NXB TON T14:52 1.0 5 0 BND EOR
% Rung: 106 %
SOR XIC B13:0/1 BST XIO I:4.0/4 NXB XIC B13:8/0 XIO I:9.0/0 BND OTE B13:8/0 EOR
% Rung: 107 %
SOR XIC B13:0/1 BST XIC O:14.0/4 XIO I:8.0/0 NXB XIC B13:11/12 XIO I:9.0/0 BND BST XIC T14:53/DN OTE B13:11/12 NXB TON T14:53 1.0 5 0 BND EOR
% Rung: 108 %
SOR XIC B13:0/1 BST XIO I:4.0/5 NXB XIC B13:8/1 XIO I:9.0/0 BND OTE B13:8/1 EOR
% Rung: 109 %
SOR XIC B13:0/1 BST XIC O:14.0/5 XIO I:8.0/1 NXB XIC B13:11/13 XIO I:9.0/0 BND BST XIC T14:54/DN OTE B13:11/13 NXB TON T14:54 1.0 5 0 BND EOR

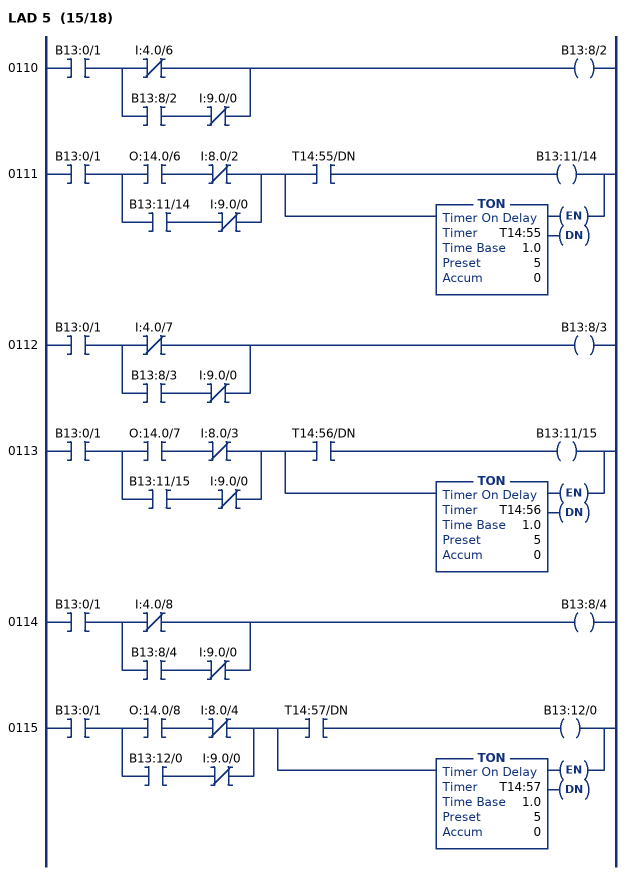
% Rung: 110 %
SOR XIC B13:0/1 BST XIO I:4.0/6 NXB XIC B13:8/2 XIO I:9.0/0 BND OTE B13:8/2 EOR
% Rung: 111 %
SOR XIC B13:0/1 BST XIC O:14.0/6 XIO I:8.0/2 NXB XIC B13:11/14 XIO I:9.0/0 BND BST XIC T14:55/DN OTE B13:11/14 NXB TON T14:55 1.0 5 0 BND EOR
% Rung: 112 %
SOR XIC B13:0/1 BST XIO I:4.0/7 NXB XIC B13:8/3 XIO I:9.0/0 BND OTE B13:8/3 EOR
% Rung: 113 %
SOR XIC B13:0/1 BST XIC O:14.0/7 XIO I:8.0/3 NXB XIC B13:11/15 XIO I:9.0/0 BND BST XIC T14:56/DN OTE B13:11/15 NXB TON T14:56 1.0 5 0 BND EOR
% Rung: 114 %
SOR XIC B13:0/1 BST XIO I:4.0/8 NXB XIC B13:8/4 XIO I:9.0/0 BND OTE B13:8/4 EOR
% Rung: 115 %
SOR XIC B13:0/1 BST XIC O:14.0/8 XIO I:8.0/4 NXB XIC B13:12/0 XIO I:9.0/0 BND BST XIC T14:57/DN OTE B13:12/0 NXB TON T14:57 1.0 5 0 BND EOR

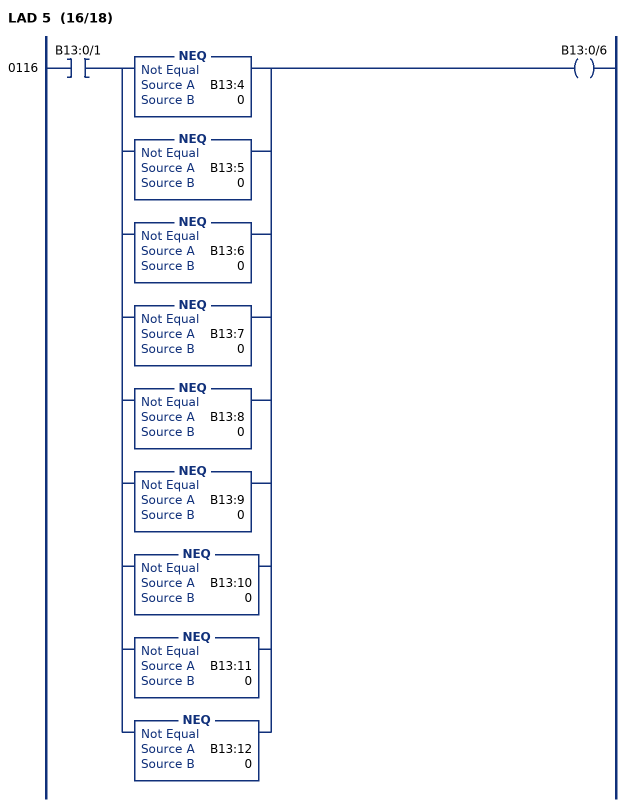
% Rung: 116 %
SOR XIC B13:0/1 BST NEQ B13:4 0 NXB NEQ B13:5 0 NXB NEQ B13:6 0 NXB NEQ B13:7 0 NXB NEQ B13:8 0 NXB NEQ B13:9 0 NXB NEQ B13:10 0 NXB NEQ B13:11 0 NXB NEQ B13:12 0 BND OTE B13:0/6 EOR

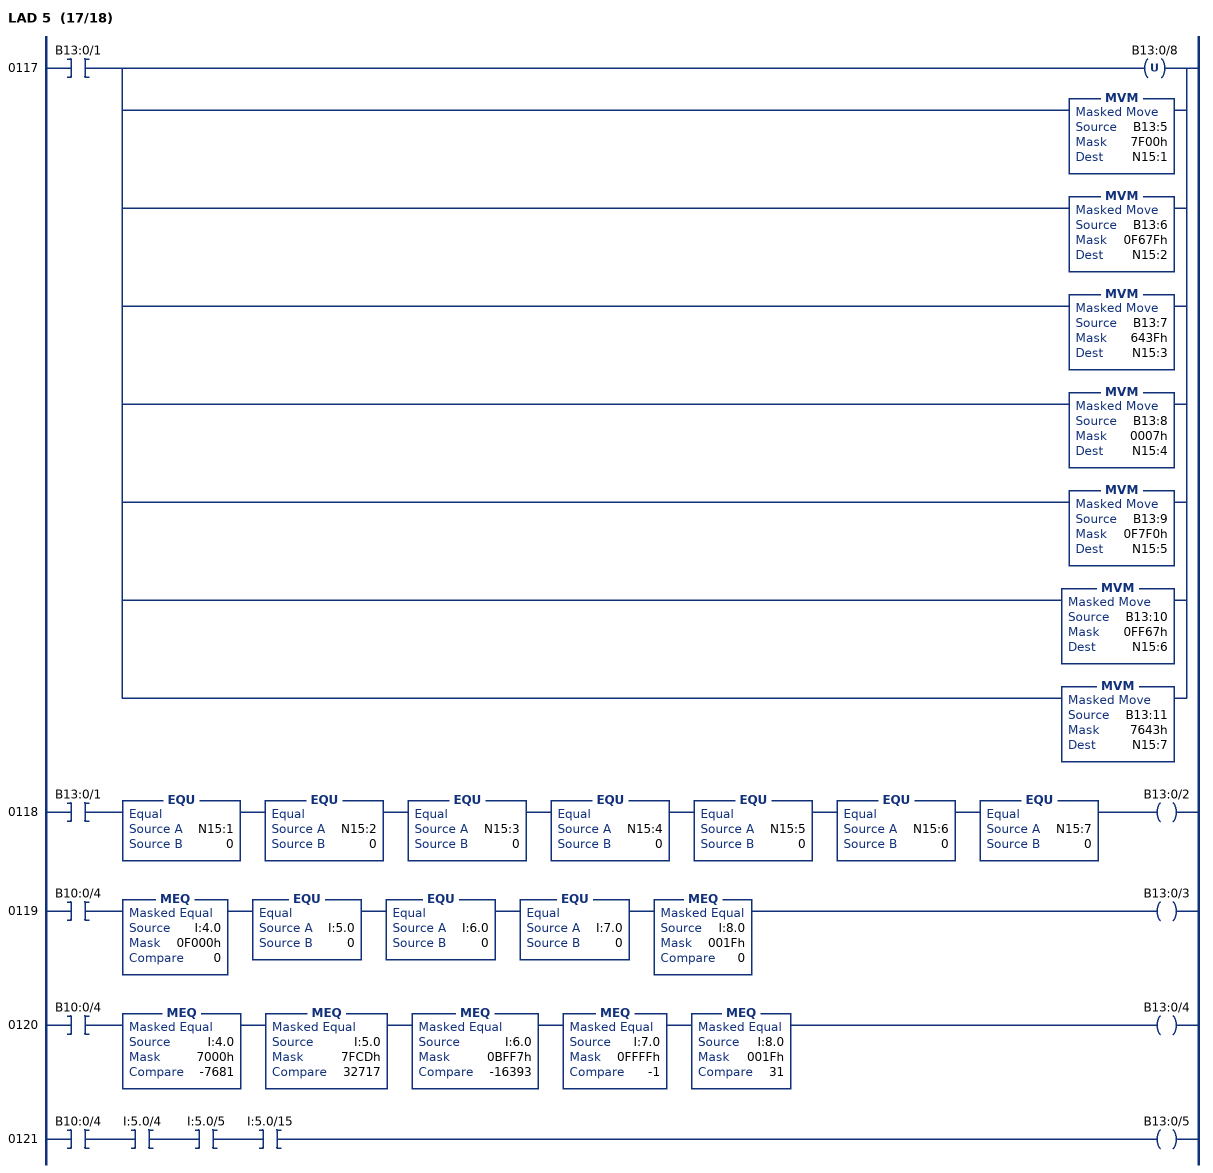
% Rung: 117 %
SOR XIC B13:0/1 BST OTU B13:0/8 NXB MVM B13:5 7F00h N15:1 NXB MVM B13:6 0F67Fh N15:2 NXB MVM B13:7 643Fh N15:3 NXB MVM B13:8 0007h N15:4 NXB MVM B13:9 0F7F0h N15:5 NXB MVM B13:10 0FF67h N15:6 NXB MVM B13:11 7643h N15:7 BND EOR
% Rung: 118 %
SOR XIC B13:0/1 EQU N15:1 0 EQU N15:2 0 EQU N15:3 0 EQU N15:4 0 EQU N15:5 0 EQU N15:6 0 EQU N15:7 0 OTE B13:0/2 EOR
% Rung: 119 %
SOR XIC B10:0/4 MEQ I:4.0 0F000h 0 EQU I:5.0 0 EQU I:6.0 0 EQU I:7.0 0 MEQ I:8.0 001Fh 0 OTE B13:0/3 EOR
% Rung: 120 %
SOR XIC B10:0/4 MEQ I:4.0 7000h -7681 MEQ I:5.0 7FCDh 32717 MEQ I:6.0 0BFF7h -16393 MEQ I:7.0 0FFFFh -1 MEQ I:8.0 001Fh 31 OTE B13:0/4 EOR
% Rung: 121 %
SOR XIC B10:0/4 XIC I:5.0/4 XIC I:5.0/5 XIC I:5.0/15 OTE B13:0/5 EOR

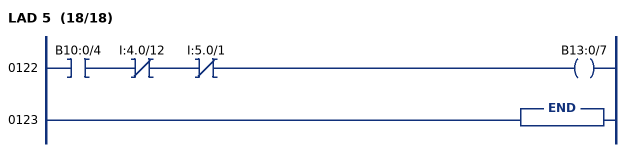
% Rung: 122 %
SOR XIC B10:0/4 XIO I:4.0/12 XIO I:5.0/1 OTE B13:0/7 EOR
% Rung: 123 %
SOR END EOR

LADDER 6
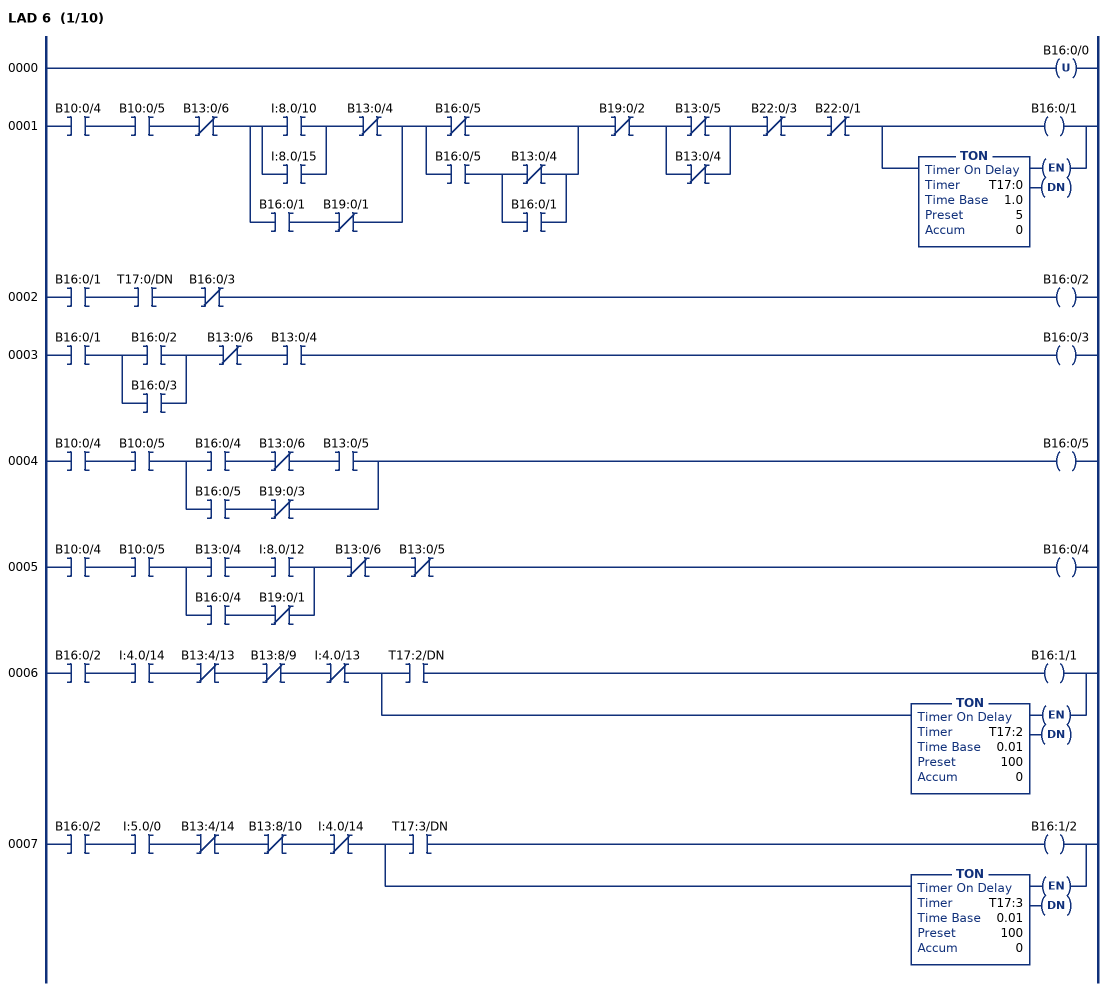
% Rung: 0 %
SOR OTU B16:0/0 EOR
% Rung: 1 %
SOR XIC B10:0/4 XIC B10:0/5 XIO B13:0/6 BST BST XIC I:8.0/10 NXB XIC I:8.0/15 BND XIO B13:0/4 NXB XIC B16:0/1 XIO B19:0/1 BND BST XIO B16:0/5 NXB XIC B16:0/5 BST XIO B13:0/4 NXB XIC B16:0/1 BND BND XIO B19:0/2 BST XIO B13:0/5 NXB XIO B13:0/4 BND XIO B22:0/3 XIO B22:0/1 BST OTE B16:0/1 NXB TON T17:0 1.0 5 0 BND EOR
% Rung: 2 %
SOR XIC B16:0/1 XIC T17:0/DN XIO B16:0/3 OTE B16:0/2 EOR
% Rung: 3 %
SOR XIC B16:0/1 BST XIC B16:0/2 NXB XIC B16:0/3 BND XIO B13:0/6 XIC B13:0/4 OTE B16:0/3 EOR
% Rung: 4 %
SOR XIC B10:0/4 XIC B10:0/5 BST XIC B16:0/4 XIO B13:0/6 XIC B13:0/5 NXB XIC B16:0/5 XIO B19:0/3 BND OTE B16:0/5 EOR
% Rung: 5 %
SOR XIC B10:0/4 XIC B10:0/5 BST XIC B13:0/4 XIC I:8.0/12 NXB XIC B16:0/4 XIO B19:0/1 BND XIO B13:0/6 XIO B13:0/5 OTE B16:0/4 EOR
% Rung: 6 %
SOR XIC B16:0/2 XIC I:4.0/14 XIO B13:4/13 XIO B13:8/9 XIO I:4.0/13 BST XIC T17:2/DN OTE B16:1/1 NXB TON T17:2 0.01 100 0 BND EOR
% Rung: 7 %
SOR XIC B16:0/2 XIC I:5.0/0 XIO B13:4/14 XIO B13:8/10 XIO I:4.0/14 BST XIC T17:3/DN OTE B16:1/2 NXB TON T17:3 0.01 100 0 BND EOR

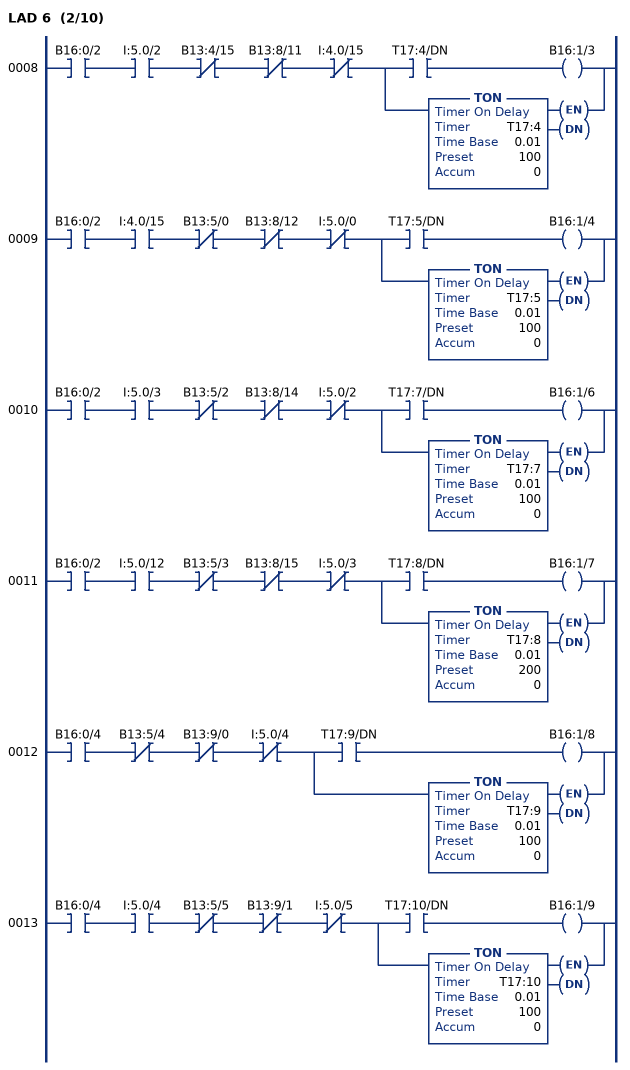
% Rung: 8 %
SOR XIC B16:0/2 XIC I:5.0/2 XIO B13:4/15 XIO B13:8/11 XIO I:4.0/15 BST XIC T17:4/DN OTE B16:1/3 NXB TON T17:4 0.01 100 0 BND EOR
% Rung: 9 %
SOR XIC B16:0/2 XIC I:4.0/15 XIO B13:5/0 XIO B13:8/12 XIO I:5.0/0 BST XIC T17:5/DN OTE B16:1/4 NXB TON T17:5 0.01 100 0 BND EOR
% Rung: 10 %
SOR XIC B16:0/2 XIC I:5.0/3 XIO B13:5/2 XIO B13:8/14 XIO I:5.0/2 BST XIC T17:7/DN OTE B16:1/6 NXB TON T17:7 0.01 100 0 BND EOR
% Rung: 11 %
SOR XIC B16:0/2 XIC I:5.0/12 XIO B13:5/3 XIO B13:8/15 XIO I:5.0/3 BST XIC T17:8/DN OTE B16:1/7 NXB TON T17:8 0.01 200 0 BND EOR
% Rung: 12 %
SOR XIC B16:0/4 XIO B13:5/4 XIO B13:9/0 XIO I:5.0/4 BST XIC T17:9/DN OTE B16:1/8 NXB TON T17:9 0.01 100 0 BND EOR
% Rung: 13 %
SOR XIC B16:0/4 XIC I:5.0/4 XIO B13:5/5 XIO B13:9/1 XIO I:5.0/5 BST XIC T17:10/DN OTE B16:1/9 NXB TON T17:10 0.01 100 0 BND EOR

